PROGRAM MAIN
VAR
	fbConsole1 : FB_ConsoleLogger;
	fbFile1 : FB_FileLogger;
	fbMachine1 : FB_Machine(fbFile1);
	fbMachine2 : FB_Machine(fbConsole1);
	
	sMessageStr1 : STRING(255):= 'This is printed in console ';
	sMessageStr2 : STRING(255) := 'This is written in file';
	
	bPass : BOOL := TRUE;
END_VAR

IF bPass THEN
	fbMachine1.M_Run(sMessageStr1);
	fbMachine2.M_Run(sMessageStr2);
	bPass := FALSE;
END_IF

END_PROGRAM

(* stored: Version 1.1.0.1, ProductVersion 3.1.4024.16
   POU MAIN: Id {50e0f26c-511e-4869-b05c-88c6177a793d}, SpecialFunc None *)
